{attribute 'qualified_only'}
VAR_GLOBAL
	Notification_ExecutionFailed : T_Notification;
	Notification_ExecutionAborted : T_Notification;
	
	
	
	
	
END_VAR

(* stored: Version 1.1.0.1, ProductVersion 3.1.4024.12
   GVL GlobalNotifications: Id {6ec84d7a-4d98-4985-8d2d-17ae6e719906} *)
